// Mitsubishi GX Works2 project: 실린더응용3   PLC: Q02/Q02H

PROGRAM MAIN
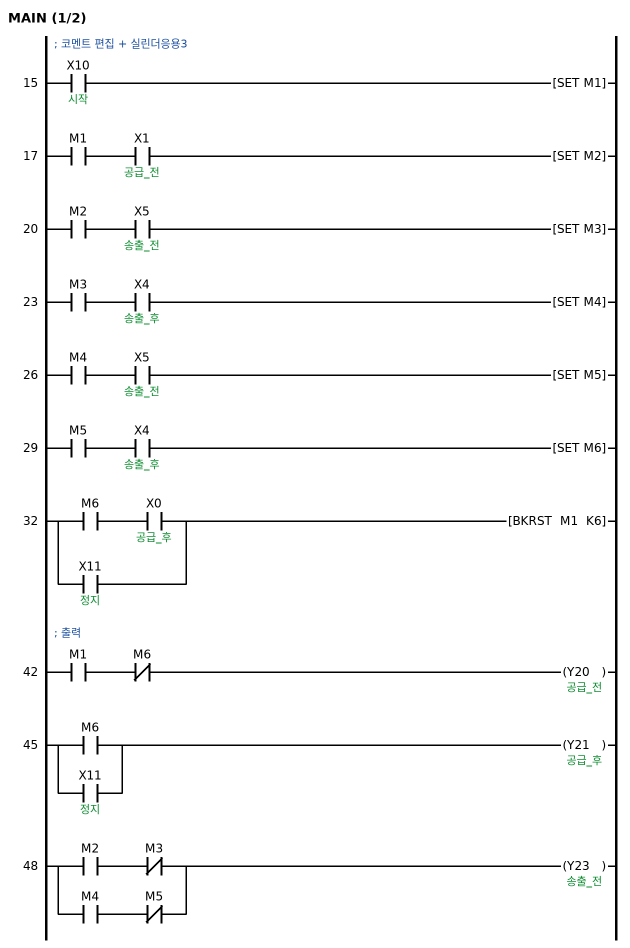
; 코멘트 편집 + 실린더응용3
15    LD      X10  ; 시작
      SET     M1
17    LD      M1
      AND     X1  ; 공급_전
      SET     M2
20    LD      M2
      AND     X5  ; 송출_전
      SET     M3
23    LD      M3
      AND     X4  ; 송출_후
      SET     M4
26    LD      M4
      AND     X5  ; 송출_전
      SET     M5
29    LD      M5
      AND     X4  ; 송출_후
      SET     M6
32    LD      M6
      AND     X0  ; 공급_후
      OR      X11  ; 정지
      BKRST   M1 K6
; 출력
42    LD      M1
      ANI     M6
      OUT     Y20  ; 공급_전
45    LD      M6
      OR      X11  ; 정지
      OUT     Y21  ; 공급_후
48    LD      M2
      ANI     M3
      LD      M4
      ANI     M5
      ORB
      OUT     Y23  ; 송출_전
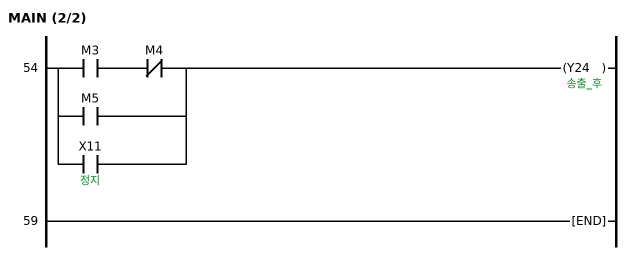
54    LD      M3
      ANI     M4
      OR      M5
      OR      X11  ; 정지
      OUT     Y24  ; 송출_후
59    END
END_PROGRAM

// device comments not shown above
X2  ; 드릴_상
X3  ; 드릴_하
X6  ; 배출_후
X7  ; 배출_전
Y22  ; 드릴_하
Y25  ; 배출_전
Y26  ; 배출_후
